(*Funzione che restituisce il numero della postazione avente una lista in lavorazione*)
FUNCTION TFWAM_RicavaListaInLavoro : UINT
VAR_INPUT
	WorkAreaProductionList : POINTER TO ARRAY [1..MAXAREA] OF TFMachinePalletizer_ListaProduzione_WAM; //Lista di produzione che devo Svolgere PER ogni POSTAZIONE
END_VAR
VAR
	i:UINT;
END_VAR

(* Ciclo tutte le Liste *)
FOR i:=1 TO MAXAREAPRESENT DO
	(* Se Lista NON è già stata avviata e NON è TERMINATA*)
	IF WorkAreaProductionList^[i].Stato >= LISTA_PROD_IN_ESECUZIONE AND WorkAreaProductionList^[i].Stato < LISTA_PROD_ESEGUITA THEN
		TFWAM_RicavaListaInLavoro := i;
		RETURN;
	END_IF
END_FOR
TFWAM_RicavaListaInLavoro:=0;

END_FUNCTION

(* stored: Version 1.1.0.1, ProductVersion 3.1.4024.11
   POU TFWAM_RicavaListaInLavoro: Id {6dbf3cf6-7f0a-491a-9cb7-298528952c04}, SpecialFunc None *)
